TYPE E_SIDEFLEX_UnitType :
(
	E_SIDEFLEX_UNKNOWN			:= 0,
	E_SIDEFLEX_2PROG				:= 1,
	E_SIDEFLEX_4PROG				:= 2
);
END_TYPE

(* stored: Version 1.1.0.1, ProductVersion 3.1.4024.15
   DUT E_SIDEFLEX_UnitType: Id {1b422683-95b1-4351-ac11-a36c5885ff95} *)
